Staubli VAL3: Kill.pgx

program Kill()
begin
  if taskStatus("readAtiForce")!=-1
    taskKill("readAtiForce")
  endIf
  //
  if taskStatus("PC_IO")!=-1
    taskKill("PC_IO")
  endIf
  if taskStatus("Input")!=-1
    taskKill("Input")
  endIf
  if taskStatus("Output")!=-1
    taskKill("Output")
  endIf
  if taskStatus("txtLoad")!=-1
    taskKill("txtLoad")
  endIf
  if taskStatus("motion")!=-1
    taskKill("motion")
  endIf
  if taskStatus("prdMassage")!=-1
    taskKill("prdMassage")
  endIf

end
